PROGRAM A02_StartupArchiveDB
VAR
	fbStartLogger: NT_StartProcess;
	fbPulse: FB_SquareWave;
	tonNotRunning: TON;
	bBusyOnce	:BOOL;

	ton_Watchdog: TON;
	nLastWatchdogFromArchiveDB	: DINT;
	bWait: BOOL;

	bArchiveDBLocalRun : BOOL;

END_VAR

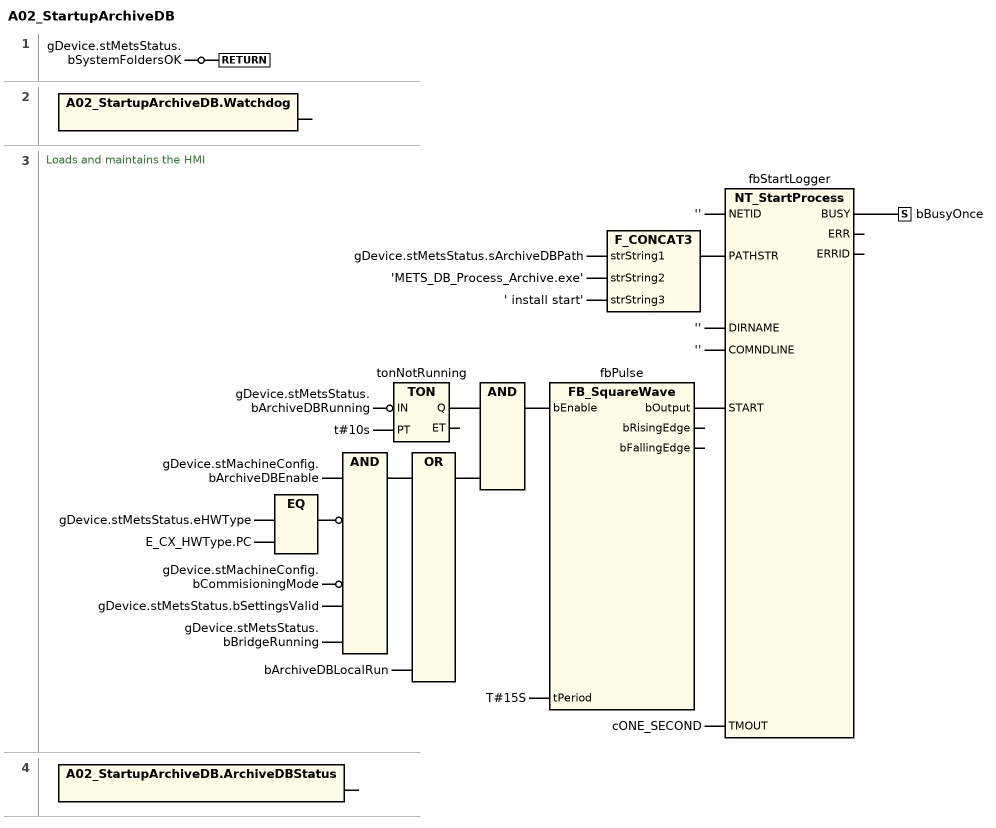
// NETWORK 1
IF NOT gDevice.stMetsStatus.bSystemFoldersOK THEN RETURN; END_IF

// NETWORK 2
A02_StartupArchiveDB.Watchdog();

// NETWORK 3
// Loads and maintains the HMI
tonNotRunning(IN := NOT gDevice.stMetsStatus.bArchiveDBRunning, PT := t#10s); // TON
fbPulse(bEnable := tonNotRunning.Q AND (gDevice.stMachineConfig.bArchiveDBEnable AND NOT (gDevice.stMetsStatus.eHWType = E_CX_HWType.PC) AND NOT gDevice.stMachineConfig.bCommisioningMode AND gDevice.stMetsStatus.bSettingsValid AND gDevice.stMetsStatus.bBridgeRunning OR bArchiveDBLocalRun), tPeriod := T#15S); // FB_SquareWave
fbStartLogger(
    NETID := '',
    PATHSTR := F_CONCAT3(strString1 := gDevice.stMetsStatus.sArchiveDBPath, strString2 := 'METS_DB_Process_Archive.exe', strString3 := ' install start'),
    DIRNAME := '',
    COMNDLINE := '',
    START := fbPulse.bOutput,
    TMOUT := cONE_SECOND); // NT_StartProcess
bBusyOnce S= fbStartLogger.BUSY;

// NETWORK 4
A02_StartupArchiveDB.ArchiveDBStatus();

ACTION ArchiveDBStatus:
(*

Initialized = 0,
HasError = 1,
UseFiles = 2,
UseDb = 3,
DbConnected = 4,
TcConnected = 5,
ApiWork = 6

*)

(*Status form SrchiveDB service*)	
gDevice.stArchiveDB.bInitialized	:= gDevice.stArchiveDB.nArchiveDBStatus.0;
gDevice.stArchiveDB.bHasError		:= gDevice.stArchiveDB.nArchiveDBStatus.1;
gDevice.stArchiveDB.bUseFiles		:= gDevice.stArchiveDB.nArchiveDBStatus.2;
gDevice.stArchiveDB.bUseDb			:= gDevice.stArchiveDB.nArchiveDBStatus.3;
gDevice.stArchiveDB.bDbConnected	:= gDevice.stArchiveDB.nArchiveDBStatus.4;
gDevice.stArchiveDB.bTcConnected	:= gDevice.stArchiveDB.nArchiveDBStatus.5;
gDevice.stArchiveDB.bApiWork		:= gDevice.stArchiveDB.nArchiveDBStatus.6;

(*Status to SrchiveDB service*)	
gDevice.stArchiveDB.bClearProdData	:= gDevice.stMetsStatus.bClearProcessFolders;		

gDevice.stArchiveDB.nMaximumCACArchiveAge	:= gDevice.stMachineConfig.nMaximumArchiveAge;
gDevice.stArchiveDB.nMaximumErrorFiles	:= gDevice.stMachineConfig.nMaximumErrorFiles;
gDevice.stArchiveDB.nMaximumOCVFiles	:= gDevice.stMachineConfig.nMaximumOCVFiles;		
gDevice.stArchiveDB.nMaximumOACFiles	:= gDevice.stMachineConfig.nMaximumOACFiles;
END_ACTION

ACTION Watchdog:
(*Watchdog to Bridge*)
gDevice.nWatchdogToArchiveDB := gDevice.nWatchdogToArchiveDB + 1;
IF  gDevice.nWatchdogToArchiveDB > 10000 THEN
	gDevice.nWatchdogToArchiveDB := 1;
END_IF

gDevice.nWatchdogFromArchiveDB	:=	gDevice.stArchiveDB.nArchiveDBWatchdog;
(*Watchdog from HMI - check if running*)
IF ton_Watchdog.Q THEN
	bWait := FALSE;
	IF gDevice.nWatchdogFromArchiveDB <> nLastWatchdogFromArchiveDB THEN
		gDevice.stMetsStatus.bArchiveDBRunning := TRUE;
		nLastWatchdogFromArchiveDB := gDevice.nWatchdogFromArchiveDB;
	ELSE
		gDevice.stMetsStatus.bArchiveDBRunning := FALSE;
	END_IF
ELSE
	bWait := TRUE;
END_IF

ton_Watchdog(IN:= bWait, PT := t#4000ms);
END_ACTION

END_PROGRAM

(* stored: Version 1.1.0.1
   POU A02_StartupArchiveDB: Id {177c7d4a-d2fc-4d88-b806-4a7fd259ef4f}, SpecialFunc None
   Action ArchiveDBStatus: Id {5f34067f-5ab3-4cca-8455-80c4aca5795a}
   Action Watchdog: Id {f98364f2-eeda-4e89-94bf-900664ab07b7} *)
